PROGRAM MAIN
VAR
END_VAR

prgECatDiag();

END_PROGRAM

(* stored: Version 1.1.0.1
   POU MAIN: Id {68b42221-f5ef-41d9-83ae-f46ca20299cf}, SpecialFunc None *)
